INTERFACE PUBLIC HoldableStateCommands EXTENDS __System.IQueryInterface

METHOD PUBLIC Hold
END_METHOD

END_INTERFACE

(* stored: Version 1.1.0.1, ProductVersion 3.1.4026.18
   Itf HoldableStateCommands: Id {045fffe5-c212-0816-1984-6a705dc8c922}
   Method Hold: Id {551ebce7-7697-0fdc-339e-d35a91bb7421} *)
